// ---- VISUs/Text/InputText.TcTLO
TEXTLIST InputText
  0 = 'IN00 启动' | Chinese: 'IN00 启动' | English: 'IN00 Start' | Vietnamese: 'IN00 Kh?i ??ng ?'
  1 = 'IN01 停止' | Chinese: 'IN01 停止' | English: 'IN01 Stop' | Vietnamese: 'IN01 D?ng l?i ?'
  2 = 'IN02 复位' | Chinese: 'IN02 复位' | English: 'IN02 ResetAlarm' | Vietnamese: 'IN02 Tuy nhiên ?'
  3 = 'IN03 急停' | Chinese: 'IN03 急停' | English: 'IN03 EStop' | Vietnamese: 'IN03 V?i d?ng l?i ?'
  4 = 'IN04 安全门开关' | Chinese: 'IN04 安全门开关' | English: 'IN04 Door' | Vietnamese: 'IN04 Chuy?n ??i c?a an toàn ?'
  5 = 'IN05 工装误合盖检测光电 ' | Chinese: 'IN05 工装误合盖检测光电 ' | English: 'IN05 FrockCloseCheck' | Vietnamese: 'IN05 FrockCloseCheck'
  6 = 'IN06 解锁站流入光电' | Chinese: 'IN06 解锁站流入光电' | English: 'IN06 OpenLockCheck0' | Vietnamese: 'IN06 OpenLockCheck0'
  7 = 'IN07 预留' | Chinese: 'IN07 预留' | English: 'IN07 None3' | Vietnamese: 'IN07 Dành riêng ?'
  8 = 'IN08 主流线拨料升降气缸原位' | Chinese: 'IN08 主流线拨料升降气缸原位' | English: 'IN08 Line0PushElevator_Cyl_H' | Vietnamese: 'IN08 Line0PushElevator_Cyl_H'
  9 = 'IN09 主流线拨料升降气缸工作位' | Chinese: 'IN09 主流线拨料升降气缸工作位' | English: 'IN09 Line0PushElevator_Cyl_W' | Vietnamese: 'IN09 Line0PushElevator_Cyl_W'
  10 = 'IN0A 预留' | Chinese: 'IN0A 预留' | English: 'IN0A None6' | Vietnamese: 'IN0A Dành riêng ?'
  11 = 'IN0B 预留' | Chinese: 'IN0B 预留' | English: 'IN0B None7' | Vietnamese: 'IN0B Dành riêng ?'
  12 = 'IN0C 主流线拨料气缸安全位' | Chinese: 'IN0C 主流线拨料气缸安全位' | English: 'IN0C Line0Push_Cyl_Safe' | Vietnamese: 'IN0C Line0Push_Cyl_Safe'
  13 = 'IN0D 接驳线前阻挡光电' | Chinese: 'IN0D 接驳线前阻挡光电' | English: 'IN0D AcquireCheck3' | Vietnamese: 'IN0D AcquireCheck3'
  14 = 'IN0E 接驳线前前阻挡气缸原位' | Chinese: 'IN0E 接驳线前前阻挡气缸原位' | English: 'IN0E AcquirePrevent2_Cyl_H' | Vietnamese: 'IN0E AcquirePrevent2_Cyl_H'
  15 = 'IN0F 接驳线前前阻挡气缸工作位' | Chinese: 'IN0F 接驳线前前阻挡气缸工作位' | English: 'IN0F AcquirePrevent2_Cyl_W' | Vietnamese: 'IN0F AcquirePrevent2_Cyl_W'
  16 = 'IN10 主流线分料气缸原位' | Chinese: 'IN10 主流线分料气缸原位' | English: 'IN10 Line0Part_Cyl_H' | Vietnamese: 'IN10 Xi lanh ph?n ph?i dòng chính ?'
  17 = 'IN11 主流线分料气缸工作位' | Chinese: 'IN11 主流线分料气缸工作位' | English: 'IN11 Line0Part_Cyl_W' | Vietnamese: 'IN11 Xi lanh làm vi?c dòng chính ?'
  18 = 'IN12 主流线阻挡气缸原位' | Chinese: 'IN12 主流线阻挡气缸原位' | English: 'IN12 Line0Prevent_Cyl_H' | Vietnamese: 'IN12 Dòng chính ch?n xi lanh ?'
  19 = 'IN13 主流线阻挡气缸工作位' | Chinese: 'IN13 主流线阻挡气缸工作位' | English: 'IN13 Line0Prevent_Cyl_W' | Vietnamese: 'IN13 Dòng chính ch?n v? trí làm vi?c c?a xi lanh ?'
  20 = 'IN14 主流线拨料气缸原位' | Chinese: 'IN14 主流线拨料气缸原位' | English: 'IN14 Line0Push_Cyl_H' | Vietnamese: 'IN14 Xi lanh ?i?u ch?nh dòng chính ?'
  21 = 'IN15 主流线拨料气缸工作位' | Chinese: 'IN15 主流线拨料气缸工作位' | English: 'IN15 Line0Push_Cyl_W' | Vietnamese: 'IN15 Xi lanh dòng chính dòng v? trí làm vi?c ?'
  22 = 'IN16 接驳线前阻挡气缸原位' | Chinese: 'IN16 接驳线前阻挡气缸原位' | English: 'IN16 AcquirePrevent0_Cyl_H' | Vietnamese: 'IN16 Ch?n xi lanh tr??c d?y n?i ?'
  23 = 'IN17 接驳线前阻挡气缸工作位' | Chinese: 'IN17 接驳线前阻挡气缸工作位' | English: 'IN17 AcquirePrevent0_Cyl_W' | Vietnamese: 'IN17 Ch?n xi lanh tr??c d?y n?i ?'
  24 = 'IN18 接驳线后阻挡气缸原位' | Chinese: 'IN18 接驳线后阻挡气缸原位' | English: 'IN18 AcquirePrevent1_Cyl_H' | Vietnamese: 'IN18 Ch?n xi lanh t?i v? trí sau khi k?t n?i ?'
  25 = 'IN19 接驳线后阻挡气缸工作位' | Chinese: 'IN19 接驳线后阻挡气缸工作位' | English: 'IN19 AcquirePrevent1_Cyl_W' | Vietnamese: 'IN19 Ch?n xi lanh sau khi k?t n?i ?'
  26 = 'IN1A 接驳线顶升气缸原位' | Chinese: 'IN1A 接驳线顶升气缸原位' | English: 'IN1A AcquireLift_Cyl_H' | Vietnamese: 'IN1A Xi lanh Leo lên d?y ?i?n v? trí ?'
  27 = 'IN1B 接驳线顶升气缸工作位' | Chinese: 'IN1B 接驳线顶升气缸工作位' | English: 'IN1B AcquireLift_Cyl_W' | Vietnamese: 'IN1B Xi lanh làm vi?c trên d?y n?i ?'
  28 = 'IN1C 接驳模组拨料气缸原位' | Chinese: 'IN1C 接驳模组拨料气缸原位' | English: 'IN1C AcquirePush_Cyl_H' | Vietnamese: 'IN1C Xi lanh kh?p n?i m?-?un v? trí ?'
  29 = 'IN1D 接驳模组拨料气缸工作位' | Chinese: 'IN1D 接驳模组拨料气缸工作位' | English: 'IN1D AcquirePush_Cyl_W' | Vietnamese: 'IN1D Xi lanh làm vi?c k?t n?i m?-?un ?'
  30 = 'IN1E 接驳模组升降气缸原位' | Chinese: 'IN1E 接驳模组升降气缸原位' | English: 'IN1E AcquireElevator_Cyl_H' | Vietnamese: 'IN1E Xi lanh n?ng m?-?un k?t n?i v? trí ?'
  31 = 'IN1F 接驳模组升降气缸工作位' | Chinese: 'IN1F 接驳模组升降气缸工作位' | English: 'IN1F AcquireElevator_Cyl_W' | Vietnamese: 'IN1F K?t n?i m?-?un n?ng xi lanh v? trí làm vi?c ?'
  32 = 'IN20 转向站顶升气缸原位' | Chinese: 'IN20 转向站顶升气缸原位' | English: 'IN20 SteeringLift_Cyl_H' | Vietnamese: 'IN20 H??ng v? v? trí xi lanh n?ng lên ?'
  33 = 'IN21 转向站顶升气缸工作位' | Chinese: 'IN21 转向站顶升气缸工作位' | English: 'IN21 SteeringLift_Cyl_W' | Vietnamese: 'IN21 V? trí làm vi?c c?a xi lanh n?ng lên ?'
  34 = 'IN22 转向站接驳升降气缸原位' | Chinese: 'IN22 转向站接驳升降气缸原位' | English: 'IN22 SteeringAcquireElevator_Cyl_H' | Vietnamese: 'IN22 Chuy?n h??ng k?t n?i v?i xi lanh n?ng t?i v? trí ?'
  35 = 'IN23 转向站接驳升降气缸工作位' | Chinese: 'IN23 转向站接驳升降气缸工作位' | English: 'IN23 SteeringAcquireElevator_Cyl_W' | Vietnamese: 'IN23 Chuy?n h??ng tr?m n?i xi lanh n?ng v? trí làm vi?c ?'
  36 = 'IN24 转向站旋转气缸原位' | Chinese: 'IN24 转向站旋转气缸原位' | English: 'IN24 SteeringRotate_Cyl_H' | Vietnamese: 'IN24 Tr?m quay quay xi lanh v? trí ?'
  37 = 'IN25 转向站旋转气缸工作位' | Chinese: 'IN25 转向站旋转气缸工作位' | English: 'IN25 SteeringRotate_Cyl_W' | Vietnamese: 'IN25 Tr?m quay quay xi lanh v? trí làm vi?c ?'
  38 = 'IN26 转向站接驳限位气缸原位' | Chinese: 'IN26 转向站接驳限位气缸原位' | English: 'IN26 SteeringAcquireLimit_Cyl_H' | Vietnamese: 'IN26 Xi lanh gi?i h?n k?t n?i tr?m lái ?'
  39 = 'IN27 转向站接驳限位气缸工作位' | Chinese: 'IN27 转向站接驳限位气缸工作位' | English: 'IN27 SteeringAcquireLimit_Cyl_W' | Vietnamese: 'IN27 V? trí làm vi?c c?a xi lanh gi?i h?n k?t n?i tr?m lái ?'
  40 = 'IN28 解锁站阻挡气缸原位' | Chinese: 'IN28 解锁站阻挡气缸原位' | English: 'IN28 OpenLockPrevent_Cyl_H' | Vietnamese: 'IN28 M? khóa tr?m ?? ng?n ch?n xi lanh ?'
  41 = 'IN29 解锁站阻挡气缸工作位' | Chinese: 'IN29 解锁站阻挡气缸工作位' | English: 'IN29 OpenLockPrevent_Cyl_W' | Vietnamese: 'IN29 M? khóa tr?m ?? ch?n v? trí làm vi?c c?a xi lanh ?'
  42 = 'IN2A 解锁站顶升气缸原位' | Chinese: 'IN2A 解锁站顶升气缸原位' | English: 'IN2A OpenLockLift_Cyl_H' | Vietnamese: 'IN2A M? khóa tr?m n?ng xi lanh v? trí ?'
  43 = 'IN2B 解锁站顶升气缸工作位' | Chinese: 'IN2B 解锁站顶升气缸工作位' | English: 'IN2B OpenLockLift_Cyl_W' | Vietnamese: 'IN2B Xi lanh m? khóa tr?m làm vi?c ?'
  44 = 'IN2C 解锁站侧推气缸原位' | Chinese: 'IN2C 解锁站侧推气缸原位' | English: 'IN2C OpenLockPush_Cyl_H' | Vietnamese: 'IN2C M? khóa xi lanh ??y ga ?'
  45 = 'IN2D 解锁站侧推气缸工作位' | Chinese: 'IN2D 解锁站侧推气缸工作位' | English: 'IN2D OpenLockPush_Cyl_W' | Vietnamese: 'IN2D M? khóa v? trí làm vi?c xi lanh ??y ga ?'
  46 = 'IN2E 解锁站旋转气缸原位' | Chinese: 'IN2E 解锁站旋转气缸原位' | English: 'IN2E OpenLockRotate_Cyl_H' | Vietnamese: 'IN2E M? khóa tr?m quay xi lanh v? trí ?'
  47 = 'IN2F 解锁站旋转气缸工作位' | Chinese: 'IN2F 解锁站旋转气缸工作位' | English: 'IN2F OpenLockRotate_Cyl_W' | Vietnamese: 'IN2F Tr?m m? khóa xi lanh quay v? trí làm vi?c ?'
  48 = 'IN30 解锁站侧推气缸2原位' | Chinese: 'IN30 解锁站侧推气缸2原位' | English: 'IN30 OpenLockPush2_Cyl_H' | Vietnamese: 'IN30 M? khóa xi lanh 2 ??y ga ?'
  49 = 'IN31 解锁站侧推气缸2工作位' | Chinese: 'IN31 解锁站侧推气缸2工作位' | English: 'IN31 OpenLockPush2_Cyl_W' | Vietnamese: 'IN31 M? khóa xi lanh bên ga ??y v? trí làm vi?c 2 ?'
  50 = 'IN32 取UC站阻挡气缸原位' | Chinese: 'IN32 取UC站阻挡气缸原位' | English: 'IN32 TakeUcPrevent_Cyl_H' | Vietnamese: 'IN32 L?y tr? UC ?? ch?n xi lanh ?'
  51 = 'IN33 取UC站阻挡气缸工作位' | Chinese: 'IN33 取UC站阻挡气缸工作位' | English: 'IN33 TakeUcPrevent_Cyl_W' | Vietnamese: 'IN33 L?y v? trí làm vi?c c?a xi lanh t? tr?m UC ?'
  52 = 'IN34 取UC站顶升气缸原位' | Chinese: 'IN34 取UC站顶升气缸原位' | English: 'IN34 TakeUcLift_Cyl_H' | Vietnamese: 'IN34 L?y xi lanh n?ng lên ? tr?m UC ?'
  53 = 'IN35 取UC站顶升气缸工作位' | Chinese: 'IN35 取UC站顶升气缸工作位' | English: 'IN35 TakeUcLift_Cyl_W' | Vietnamese: 'IN35 L?y v? trí làm vi?c c?a xi lanh n?ng lên t? tr?m UC ?'
  54 = 'IN36 取UC站侧推气缸原位' | Chinese: 'IN36 取UC站侧推气缸原位' | English: 'IN36 TakeUcPush_Cyl_H' | Vietnamese: 'IN36 L?y xi lanh ??y bên ga UC ?'
  55 = 'IN37 取UC站侧推气缸工作位' | Chinese: 'IN37 取UC站侧推气缸工作位' | English: 'IN37 TakeUcPush_Cyl_W' | Vietnamese: 'IN37 L?y v? trí làm vi?c c?a xi lanh ??y bên ga UC ?'
  56 = 'IN38 取UC站旋转气缸原位' | Chinese: 'IN38 取UC站旋转气缸原位' | English: 'IN38 TakeUcRotate_Cyl_H' | Vietnamese: 'IN38 L?y xi lanh quay ? tr?m UC ?'
  57 = 'IN39 取UC站旋转气缸工作位' | Chinese: 'IN39 取UC站旋转气缸工作位' | English: 'IN39 TakeUcRotate_Cyl_W' | Vietnamese: 'IN39 L?y v? trí quay xi lanh c?a tr?m UC ?'
  58 = 'IN3A 取UC站校平气缸原位' | Chinese: 'IN3A 取UC站校平气缸原位' | English: 'IN3A TakeUcStandard_Cyl_H' | Vietnamese: 'IN3A L?y xi lanh ph?ng ? ga UC ?'
  59 = 'IN3B 取UC站校平气缸工作位' | Chinese: 'IN3B 取UC站校平气缸工作位' | English: 'IN3B TakeUcStandard_Cyl_W' | Vietnamese: 'IN3B Tr?m ki?m tra xi lanh b?ng ph?ng ?'
  60 = 'IN3C 取UC站工装夹紧气缸原位' | Chinese: 'IN3C 取UC站工装夹紧气缸原位' | English: 'IN3C TakeUcFrockClamp_Cyl_H' | Vietnamese: 'IN3C L?y xi lanh k?p vào v? trí c?a tr?m UC'
  61 = 'IN3D 取UC站工装夹紧气缸工作位' | Chinese: 'IN3D 取UC站工装夹紧气缸工作位' | English: 'IN3D TakeUcFrockClamp_Cyl_W' | Vietnamese: 'IN3D L?y v? trí làm vi?c xi lanh cài ??t ? ga UC'
  62 = 'IN3E 下工装站阻挡气缸原位' | Chinese: 'IN3E 下工装站阻挡气缸原位' | English: 'IN3E UnloadFrockPrevent_Cyl_H' | Vietnamese: 'IN3E Ng?n ch?n xi lanh ? v? trí c?ng c? ?'
  63 = 'IN3F 下工装站阻挡气缸工作位' | Chinese: 'IN3F 下工装站阻挡气缸工作位' | English: 'IN3F UnloadFrockPrevent_Cyl_W' | Vietnamese: 'IN3F Tr?m d?ng xi lanh làm vi?c ?'
  64 = 'IN40 下工装站顶升气缸原位' | Chinese: 'IN40 下工装站顶升气缸原位' | English: 'IN40 UnloadFrockLift_Cyl_H' | Vietnamese: 'IN40 Xi lanh n?ng lên xu?ng ga v? trí ?'
  65 = 'IN41 下工装站顶升气缸工作位' | Chinese: 'IN41 下工装站顶升气缸工作位' | English: 'IN41 UnloadFrockLift_Cyl_W' | Vietnamese: 'IN41 Xi lanh n?ng lên các tr?m làm vi?c ?'
  66 = 'IN42 下工装站拨料气缸原位' | Chinese: 'IN42 下工装站拨料气缸原位' | English: 'IN42 UnloadFrockPush_Cyl_H' | Vietnamese: 'IN42 Xi lanh xi lanh ? v? trí ti?p theo ?'
  67 = 'IN43 下工装站拨料气缸工作位' | Chinese: 'IN43 下工装站拨料气缸工作位' | English: 'IN43 UnloadFrockPush_Cyl_W' | Vietnamese: 'IN43 Xi lanh theo tr?m làm vi?c ?'
  68 = 'IN44 取UC模组平移Y气缸原位' | Chinese: 'IN44 取UC模组平移Y气缸原位' | English: 'IN44 TakeUc1Y_Cyl_H' | Vietnamese: 'IN44 L?y m?-?un UC và chuy?n xi lanh Y vào v? trí ?'
  69 = 'IN45 取UC模组平移Y气缸工作位' | Chinese: 'IN45 取UC模组平移Y气缸工作位' | English: 'IN45 TakeUc1Y_Cyl_W' | Vietnamese: 'IN45 Thay ??i xi lanh Y b?ng m?-?un UC ?'
  70 = 'IN46 取UC模组升降Z1气缸原位' | Chinese: 'IN46 取UC模组升降Z1气缸原位' | English: 'IN46 TakeUc1Z1_Cyl_H' | Vietnamese: 'IN46 N?ng xi lanh Z1 b?ng m?-?un UC ?'
  71 = 'IN47 取UC模组升降Z1气缸工作位' | Chinese: 'IN47 取UC模组升降Z1气缸工作位' | English: 'IN47 TakeUc1Z1_Cyl_W' | Vietnamese: 'IN47 L?y m?-?un n?ng xi lanh Z1 ?'
  72 = 'IN48 取UC模组升降Z2气缸原位' | Chinese: 'IN48 取UC模组升降Z2气缸原位' | English: 'IN48 TakeUc1Z2_Cyl_H' | Vietnamese: 'IN48 L?y m?-?un UC n?ng xi lanh Z2 ?'
  73 = 'IN49 取UC模组升降Z2气缸工作位' | Chinese: 'IN49 取UC模组升降Z2气缸工作位' | English: 'IN49 TakeUc1Z2_Cyl_W' | Vietnamese: 'IN49 L?y m?-?un UC n?ng xi lanh Z2 v? trí làm vi?c ?'
  74 = 'IN4A 取UC模组旋转气缸原位' | Chinese: 'IN4A 取UC模组旋转气缸原位' | English: 'IN4A TakeUc1Rotate_Cyl_H' | Vietnamese: 'IN4A L?y xi lanh quay c?a m?-?un UC ?'
  75 = 'IN4B 取UC模组旋转气缸工作位' | Chinese: 'IN4B 取UC模组旋转气缸工作位' | English: 'IN4B TakeUc1Rotate_Cyl_W' | Vietnamese: 'IN4B L?y v? trí làm vi?c c?a xi lanh xoay m?-?un UC ?'
  76 = 'IN4C 取UC模组夹紧气缸原位' | Chinese: 'IN4C 取UC模组夹紧气缸原位' | English: 'IN4C TakeUc1Clamp_Cyl_H' | Vietnamese: 'IN4C L?y m?-?un UC k?p xi lanh vào v? trí ?'
  77 = 'IN4D 取UC模组夹紧气缸工作位' | Chinese: 'IN4D 取UC模组夹紧气缸工作位' | English: 'IN4D TakeUc1Clamp_Cyl_W' | Vietnamese: 'IN4D L?y m?-?un UC k?p xi lanh vào v? trí làm vi?c ?'
  78 = 'IN4E 下UC皮带升降气缸原位' | Chinese: 'IN4E 下UC皮带升降气缸原位' | English: 'IN4E UnloadUcElevator_Cyl_H' | Vietnamese: 'IN4E Xi lanh n?ng d??i vành ?ai UC ?'
  79 = 'IN4F 下UC皮带升降气缸工作位' | Chinese: 'IN4F 下UC皮带升降气缸工作位' | English: 'IN4F UnloadUcElevator_Cyl_W' | Vietnamese: 'IN4F V? trí làm vi?c c?a xi lanh n?ng d??i vành ?ai UC ?'
  80 = 'IN50 下UC皮带拨料气缸原位' | Chinese: 'IN50 下UC皮带拨料气缸原位' | English: 'IN50 UnloadUcConveyorPush_Cyl_H' | Vietnamese: 'IN50 Xi lanh ?i?u ch?nh d??i vành ?ai UC ?'
  81 = 'IN51 下UC皮带拨料气缸工作位' | Chinese: 'IN51 下UC皮带拨料气缸工作位' | English: 'IN51 UnloadUcConveyorPush_Cyl_W' | Vietnamese: 'IN51 Xi lanh làm vi?c d??i vành ?ai UC ?'
  82 = 'IN52 下工装皮带升降气缸原位' | Chinese: 'IN52 下工装皮带升降气缸原位' | English: 'IN52 UnloadFrockConveyorPrevent_Cyl_H' | Vietnamese: 'IN52 D?y chuy?n n?ng xi lanh cài ??t ?'
  83 = 'IN53 下工装皮带升降气缸工作位' | Chinese: 'IN53 下工装皮带升降气缸工作位' | English: 'IN53 UnloadFrockConveyorPrevent_Cyl_W' | Vietnamese: 'IN53 D?y chuy?n n?ng xi lanh làm vi?c ?'
  84 = 'IN54 下工装皮带拨料气缸原位' | Chinese: 'IN54 下工装皮带拨料气缸原位' | English: 'IN54 UnloadFrockConveyorPush_Cyl_H' | Vietnamese: 'IN54 Xi lanh d?y chuy?n theo v? trí ?'
  85 = 'IN55 下工装皮带拨料气缸工作位' | Chinese: 'IN55 下工装皮带拨料气缸工作位' | English: 'IN55 UnloadFrockConveyorPush_Cyl_W' | Vietnamese: 'IN55 Xi lanh d?y chuy?n làm vi?c ?'
  86 = 'IN56 解锁站解压侧推气缸原位' | Chinese: 'IN56 解锁站解压侧推气缸原位' | English: 'IN56 OpenLockPressPush_Cyl_H' | Vietnamese: 'IN56 OpenLockPressPush_Cyl_H'
  87 = 'IN57 解锁站解压侧推气缸工作位' | Chinese: 'IN57 解锁站解压侧推气缸工作位' | English: 'IN57 OpenLockPressPush_Cyl_W' | Vietnamese: 'IN57 OpenLockPressPush_Cyl_W'
  88 = 'IN58 解锁站解压旋转气缸原位' | Chinese: 'IN58 解锁站解压旋转气缸原位' | English: 'IN58 OpenLockPressRotate_Cyl_H' | Vietnamese: 'IN58 OpenLockPressRotate_Cyl_H'
  89 = 'IN59 解锁站解压旋转气缸工作位' | Chinese: 'IN59 解锁站解压旋转气缸工作位' | English: 'IN59 OpenLockPressRotate_Cyl_W' | Vietnamese: 'IN59 OpenLockPressRotate_Cyl_W'
  90 = 'IN5A 预留' | Chinese: 'IN5A 预留' | English: 'IN5A None34' | Vietnamese: 'IN5A Dành riêng ?'
  91 = 'IN5B 预留' | Chinese: 'IN5B 预留' | English: 'IN5B None35' | Vietnamese: 'IN5B Dành riêng ?'
  92 = 'IN5C 下UC皮带翻转气缸缩回' | Chinese: 'IN5C 下UC皮带翻转气缸缩回' | English: 'IN5C UnloadUcBeltTipper_Cyl_H' | Vietnamese: 'IN5C Quay ng??c xi lanh l?i ?'
  93 = 'IN5D 下UC皮带翻转气缸伸出' | Chinese: 'IN5D 下UC皮带翻转气缸伸出' | English: 'IN5D UnloadUcBeltTipper_Cyl_W' | Vietnamese: 'IN5D Cái xi lanh xoay d??i vành ?ai UC thò ra ?'
  94 = 'IN5E 下UC皮带顶升气缸缩回' | Chinese: 'IN5E 下UC皮带顶升气缸缩回' | English: 'IN5E UnloadUcBeltLift_Cyl_H' | Vietnamese: 'IN5E Co l?i xi lanh n?ng lên d??i vành ?ai UC ?'
  95 = 'IN5F 下UC皮带顶升气缸伸出' | Chinese: 'IN5F 下UC皮带顶升气缸伸出' | English: 'IN5F UnloadUcBeltLift_Cyl_W' | Vietnamese: 'IN5F Cái xi lanh n?ng lên d??i vành ?ai UC thò ra ?'
  96 = 'IN60 主流线分料光电' | Chinese: 'IN60 主流线分料光电' | English: 'IN60 Line0Check1' | Vietnamese: 'IN60 Dòng chính ph?n ph?i quang ?i?n ?'
  97 = 'IN61 主流线阻挡光电' | Chinese: 'IN61 主流线阻挡光电' | English: 'IN61 Line0Check2' | Vietnamese: 'IN61 Dòng chính ng?n ch?n quang ?i?n ?'
  98 = 'IN62 主流线到位光电' | Chinese: 'IN62 主流线到位光电' | English: 'IN62 Line0Check3' | Vietnamese: 'IN62 Dòng chính vào v? trí quang ?i?n ?'
  99 = 'IN63 接驳线流入光电' | Chinese: 'IN63 接驳线流入光电' | English: 'IN63 AcquireCheck1' | Vietnamese: 'IN63 ???ng d?n d?n vào quang ?i?n ?'
  100 = 'IN64 接驳线到位光电' | Chinese: 'IN64 接驳线到位光电' | English: 'IN64 AcquireCheck2' | Vietnamese: 'IN64 K?t n?i ??n v? trí quang ?i?n ?'
  101 = 'IN65 转向站到位光电' | Chinese: 'IN65 转向站到位光电' | English: 'IN65 SteeringCheck1' | Vietnamese: 'IN65 Chuy?n sang v? trí quang ?i?n ?'
  102 = 'IN66 解锁站到位光电' | Chinese: 'IN66 解锁站到位光电' | English: 'IN66 OpenLockCheck' | Vietnamese: 'IN66 M? khóa v? trí quang ?i?n ?'
  103 = 'IN67 取UC站到位光电' | Chinese: 'IN67 取UC站到位光电' | English: 'IN67 TakeUcCheck1' | Vietnamese: 'IN67 Cho tr?m n?ng l??ng m?t tr?i vào v? trí ?'
  104 = 'IN68 下工装站到位光电' | Chinese: 'IN68 下工装站到位光电' | English: 'IN68 UnloadFrockCheck1' | Vietnamese: 'IN68 Thi?t b? ??t t?i v? trí quang ?i?n ?'
  105 = 'IN69 下UC皮带流入光电' | Chinese: 'IN69 下UC皮带流入光电' | English: 'IN69 UnloadUcCheck1' | Vietnamese: 'IN69 Vành ?ai d??i UC ?ang ch?y vào quang ?i?n ?'
  106 = 'IN6A 下UC皮带到位光电' | Chinese: 'IN6A 下UC皮带到位光电' | English: 'IN6A UnloadUcCheck2' | Vietnamese: 'IN6A Phía d??i vành ?ai n?ng l??ng m?t tr?i ?'
  107 = 'IN6B 下工装站流入光电' | Chinese: 'IN6B 下工装站流入光电' | English: 'IN6B UnloadFrockStationCheck1' | Vietnamese: 'IN6B Vành ?ai c?ng c? ch?y vào quang ?i?n ?'
  108 = 'IN6C 下工装皮带到位光电' | Chinese: 'IN6C 下工装皮带到位光电' | English: 'IN6C UnloadFrockConveyorCheck2' | Vietnamese: 'IN6C Vành ?ai c?ng c? ? v? trí quang ?i?n ?'
  109 = 'IN6D 下uc皮带翻转光电' | Chinese: 'IN6D 下uc皮带翻转光电' | English: 'IN6D UnloadUcBeltTipper' | Vietnamese: 'IN6D ??o ng??c n?ng l??ng m?t tr?i ?'
  110 = 'IN6E 取UC站流入光电' | Chinese: 'IN6E 取UC站流入光电' | English: 'IN6E TakeUcCheck0' | Vietnamese: 'IN6E TakeUcCheck0'
  111 = 'IN6F 取UC模组平移Y气缸安全位' | Chinese: 'IN6F 取UC模组平移Y气缸安全位' | English: 'IN6F TakeUc1Y_Cyl_Safe' | Vietnamese: 'IN6F Dành riêng ?'
  112 = 'IN70 解锁站升降气缸原位' | Chinese: 'IN70 解锁站升降气缸原位' | English: 'IN70 OpenLockElevator_Cyl_H' | Vietnamese: 'IN70 M? khóa tr?m n?ng xi lanh v? trí ?'
  113 = 'IN71 解锁站升降气缸工作位' | Chinese: 'IN71 解锁站升降气缸工作位' | English: 'IN71 OpenLockElevator_Cyl_W' | Vietnamese: 'IN71 M? khóa tr?m n?ng xi lanh v? trí làm vi?c ?'
  114 = 'IN72 解锁站解锁平移原位' | Chinese: 'IN72 解锁站解锁平移原位' | English: 'IN72 OpenLockPin_Cyl_H' | Vietnamese: 'IN72 Tr?m m? khóa m? khóa chuy?n v? trí ?'
  115 = 'IN73 解锁站解锁平移工作位' | Chinese: 'IN73 解锁站解锁平移工作位' | English: 'IN73 OpenLockPin_Cyl_W' | Vietnamese: 'IN73 Tr?m m? khóa m? khóa chuy?n v? trí làm vi?c ?'
  116 = 'IN74 解锁站按压气缸到原位' | Chinese: 'IN74 解锁站按压气缸到原位' | English: 'IN74 TakeUcElevator_Cyl_H' | Vietnamese: 'IN74 M? khóa tr?m nh?n xi lanh vào v? trí ?'
  117 = 'IN75 解锁站按压气缸到工作位' | Chinese: 'IN75 解锁站按压气缸到工作位' | English: 'IN75 TakeUcElevator_Cyl_W' | Vietnamese: 'IN75 M? khóa tr?m nh?n xi lanh ??n v? trí làm vi?c ?'
  118 = 'IN76 取UC站升降气缸原位' | Chinese: 'IN76 取UC站升降气缸原位' | English: 'IN76 TakeUcPush1_Cyl_H' | Vietnamese: 'IN76 L?y xi lanh n?ng t? tr?m UC ?'
  119 = 'IN77 取UC站升降气缸工作位' | Chinese: 'IN77 取UC站升降气缸工作位' | English: 'IN77 TakeUcPush1_Cyl_W' | Vietnamese: 'IN77 Tr? UC n?ng xi lanh v? trí làm vi?c ?'
  120 = 'IN78 取UC站侧推1气缸到原位' | Chinese: 'IN78 取UC站侧推1气缸到原位' | English: 'IN78 None45' | Vietnamese: 'IN78 L?y ga UC ??y 1 xi lanh vào v? trí ?'
  121 = 'IN79 取UC站侧推1气缸到工作位' | Chinese: 'IN79 取UC站侧推1气缸到工作位' | English: 'IN79 None46' | Vietnamese: 'IN79 L?y ga bên ??y 1 xi lanh t?i v? trí làm vi?c ?'
  122 = 'IN7A 预留' | Chinese: 'IN7A 预留' | English: 'IN7A None45' | Vietnamese: 'IN7A Dành riêng ?'
  123 = 'IN7B 预留' | Chinese: 'IN7B 预留' | English: 'IN7B None46' | Vietnamese: 'IN7B Dành riêng ?'
  124 = 'IN7C 预留' | Chinese: 'IN7C 预留' | English: 'IN7C None47' | Vietnamese: 'IN7C Dành riêng ?'
  125 = 'IN7D 预留' | Chinese: 'IN7D 预留' | English: 'IN7D None48' | Vietnamese: 'IN7D Dành riêng ?'
  126 = 'IN7E 预留' | Chinese: 'IN7E 预留' | English: 'IN7E None49' | Vietnamese: 'IN7E Dành riêng ?'
  127 = 'IN7F 预留' | Chinese: 'IN7F 预留' | English: 'IN7F None50' | Vietnamese: 'IN7F Dành riêng ?'
   = ''
END_TEXTLIST

// ---- VISUs/Text/LineLoadClose.TcTLO
TEXTLIST LineLoadClose
  0 = '主流线&缓存线上料' | Chinese: '主流线&缓存线上料' | English: 'LineLoad_None' | Vietnamese: 'LineLoad_None'
  1 = '主流线上料关闭' | Chinese: '主流线上料关闭' | English: 'Line0Close' | Vietnamese: 'Line1Close'
  2 = '缓存线上料关闭' | Chinese: '缓存线上料关闭' | English: 'LineAcquireClose' | Vietnamese: 'LineAcquireClose'
   = ''
END_TEXTLIST

// ---- VISUs/Text/LineLoadClase.TcTLO
TEXTLIST LineLoadClase
  0 = '不选择' | Chinese: '不选择' | English: 'None' | Vietnamese: 'None'
  1 = '优先主流线' | Chinese: '优先主流线' | English: 'Priority Line0' | Vietnamese: 'Priority Line0'
  2 = '优先接驳站' | Chinese: '优先接驳站' | English: 'Priority Acquire' | Vietnamese: 'Priority Acquire'
  3 = '优先传感器' | Chinese: '优先传感器' | English: 'Priority Sensor' | Vietnamese: 'Priority Sensor'
   = ''
END_TEXTLIST

// ---- VISUs/Text/LoadPriority.TcTLO
TEXTLIST LoadPriority
  0 = 'LoadPriority_None'
  1 = 'LoadPriority_Line0'
  2 = 'LoadPriority_Line1'
   = ''
END_TEXTLIST

// ---- VISUs/Text/MachineType.TcTLO
TEXTLIST MachineType
  0 = 'None'
  1 = '367' | Chinese: '367' | English: '367' | Vietnamese: '367'
  2 = '201' | Chinese: '201' | English: '201' | Vietnamese: '201'
  3 = '373' | Chinese: '373' | English: '373' | Vietnamese: '373'
  4 = '69' | Chinese: '69' | English: '69' | Vietnamese: '69'
  5 = '311' | Chinese: '311' | English: '311' | Vietnamese: '311'
   = ''
END_TEXTLIST

// ---- VISUs/Text/ProductType.TcTLO
TEXTLIST ProductType
  0 = '无' | Chinese: '无' | English: 'None' | Vietnamese: 'None'
  1 = '左线' | Chinese: '左线' | English: 'Left' | Vietnamese: 'Left'
  2 = '右线' | Chinese: '右线' | English: 'Right' | Vietnamese: 'Right'
   = ''
END_TEXTLIST

// ---- VISUs/Text/ManualText.TcTLO
TEXTLIST ManualText
  0 = ' \n  取料Y轴\n1:初始位 2:Line0取料位 3:Line1取料位 4:Line3取料位\n\n   取料Z轴\n1:上升位 2:下降位_Line0 3:下降位_Line1\n\n   下UC_Y轴\n1:初始位 2:Line2取料位 3:Line3取料位 4:下UC位' | Chinese: ' \n  取料Y轴\n1:初始位 2:Line0取料位 3:Line1取料位 4:Line3取料位\n\n   取料Z轴\n1:上升位 2:下降位_Line0 3:下降位_Line1\n\n   下UC_Y轴\n1:初始位 2:Line2取料位 3:Line3取料位 4:下UC位' | English: ' \nPick the y axis\nThe initial bit is the initial bit 2:line0\n\nPick the z axis\nDrop _line0 3: drop _line1\n\nThe lower uc_y axis\n1: the initial bit 2:line2 takes the material bit \n3:line3 takes the material bit 4: the lower uc bit' | Vietnamese: ' \nL?y v?t li?u trên tr?c Y\n1: ban ??u bit 2: dòng 0 c?p 3: dòng 1 c?p 4: dòng 3 c?p\n\nL?y tr?c Z\n1: n?ng lên 2: h? xu?ng bit _dòng 0 3: h? xu?ng bit _dòng 1\n\nTr?c d??i UC_Y\n1: b?t ??u bit 2: dòng 2 c?p 3: dòng 3 c?p 4: UC'
   = ''
END_TEXTLIST

// ---- VISUs/Text/OutputText.TcTLO
TEXTLIST OutputText
  0 = 'OUT00 三色灯红' | Chinese: 'OUT00 三色灯红' | English: 'OUT00 Beacon_Red' | Vietnamese: 'OUT00 ?èn ?? ba màu ?'
  1 = 'OUT01 三色灯黄' | Chinese: 'OUT01 三色灯黄' | English: 'OUT01 Beacon_Yellow' | Vietnamese: 'OUT01 ?èn màu vàng ?'
  2 = 'OUT02 三色灯绿' | Chinese: 'OUT02 三色灯绿' | English: 'OUT02 Beacon_Green' | Vietnamese: 'OUT02 Màu xanh lá c?y ?èn ba màu ?'
  3 = 'OUT03 蜂鸣器' | Chinese: 'OUT03 蜂鸣器' | English: 'OUT03 Beacon_Buzzer' | Vietnamese: 'OUT03 buzzer ?'
  4 = 'OUT04 运行指示灯' | Chinese: 'OUT04 运行指示灯' | English: 'OUT04 Runing' | Vietnamese: 'OUT04 Ch?y ánh sáng ?'
  5 = 'OUT05 停止指示灯' | Chinese: 'OUT05 停止指示灯' | English: 'OUT05 Stop' | Vietnamese: 'OUT05 D?ng ?èn ?'
  6 = 'OUT06 照明灯' | Chinese: 'OUT06 照明灯' | English: 'OUT06 LED' | Vietnamese: 'OUT06 ?nh sáng ?'
  7 = 'OUT07 预留' | Chinese: 'OUT07 预留' | English: 'OUT07 None1' | Vietnamese: 'OUT07 Dành riêng ?'
  8 = 'OUT08 解锁站解压侧推气缸到原位' | Chinese: 'OUT08 解锁站解压侧推气缸到原位' | English: 'OUT08 OpenLockPressPush_Cyl_H' | Vietnamese: 'OUT08 OpenLockPressPush_Cyl_H'
  9 = 'OUT09 解锁站解压侧推气缸到工作位' | Chinese: 'OUT09 解锁站解压侧推气缸到工作位' | English: 'OUT09 OpenLockPressPush_Cyl_W' | Vietnamese: 'OUT09 OpenLockPressPush_Cyl_W'
  10 = 'OUT0A 解锁站解压旋转气缸到原位' | Chinese: 'OUT0A 解锁站解压旋转气缸到原位' | English: 'OUT0A OpenLockPressRotate_Cyl_H' | Vietnamese: 'OUT0A OpenLockPressRotate_Cyl_H'
  11 = 'OUT0B 解锁站解压旋转气缸到工作位' | Chinese: 'OUT0B 解锁站解压旋转气缸到工作位' | English: 'OUT0B OpenLockPressRotate_Cyl_W' | Vietnamese: 'OUT0B OpenLockPressRotate_Cyl_W'
  12 = 'OUT0C 主流线拨料升降气缸到原位' | Chinese: 'OUT0C 主流线拨料升降气缸到原位' | English: 'OUT0C Line0PushElevator_Cyl_H' | Vietnamese: 'OUT0C Line0PushElevator_Cyl_H'
  13 = 'OUT0D 主流线拨料升降气缸到工作位' | Chinese: 'OUT0D 主流线拨料升降气缸到工作位' | English: 'OUT0D Line0PushElevator_Cyl_W' | Vietnamese: 'OUT0D Line0PushElevator_Cyl_W'
  14 = 'OUT0E 接驳线前前阻挡气缸缩回' | Chinese: 'OUT0E 接驳线前前阻挡气缸缩回' | English: 'OUT0E AcquirePrevent2_Cyl_H' | Vietnamese: 'OUT0E AcquirePrevent2_Cyl_H'
  15 = 'OUT0F 接驳线前前阻挡气缸伸出' | Chinese: 'OUT0F 接驳线前前阻挡气缸伸出' | English: 'OUT0F AcquirePrevent2_Cyl_W' | Vietnamese: 'OUT0F AcquirePrevent2_Cyl_W'
  16 = 'OUT10 主流线分料气缸缩回' | Chinese: 'OUT10 主流线分料气缸缩回' | English: 'OUT10 Line0Part_Cyl_H' | Vietnamese: 'OUT10 Xi lanh c?a dòng chính rút lui ?'
  17 = 'OUT11 主流线分料气缸伸出' | Chinese: 'OUT11 主流线分料气缸伸出' | English: 'OUT11 Line0Part_Cyl_W' | Vietnamese: 'OUT11 Xi lanh dòng chính ra ngoài ?'
  18 = 'OUT12 主流线阻挡气缸缩回' | Chinese: 'OUT12 主流线阻挡气缸缩回' | English: 'OUT12 Line0Prevent_Cyl_H' | Vietnamese: 'OUT12 Dòng chính ng?n ch?n s? rút l?i c?a xi lanh ?'
  19 = 'OUT13 主流线阻挡气缸伸出' | Chinese: 'OUT13 主流线阻挡气缸伸出' | English: 'OUT13 Line0Prevent_Cyl_W' | Vietnamese: 'OUT13 Dòng chính ng?n các xi lanh thoát ra ?'
  20 = 'OUT14 主流线拨料气缸缩回' | Chinese: 'OUT14 主流线拨料气缸缩回' | English: 'OUT14 Line0Push_Cyl_H' | Vietnamese: 'OUT14 Xi lanh quay dòng chính rút lui ?'
  21 = 'OUT15 主流线拨料气缸伸出' | Chinese: 'OUT15 主流线拨料气缸伸出' | English: 'OUT15 Line0Push_Cyl_W' | Vietnamese: 'OUT15 Xi lanh cu?n dòng chính thò ra ?'
  22 = 'OUT16 接驳线前阻挡气缸缩回' | Chinese: 'OUT16 接驳线前阻挡气缸缩回' | English: 'OUT16 AcquirePrevent0_Cyl_H' | Vietnamese: 'OUT16 Khóa xi lanh tr??c d?y n?i rút l?i ?'
  23 = 'OUT17 接驳线前阻挡气缸伸出' | Chinese: 'OUT17 接驳线前阻挡气缸伸出' | English: 'OUT17 AcquirePrevent0_Cyl_W' | Vietnamese: 'OUT17 Ch?n xi lanh tr??c d?y n?i ?'
  24 = 'OUT18 接驳线后阻挡气缸缩回' | Chinese: 'OUT18 接驳线后阻挡气缸缩回' | English: 'OUT18 AcquirePrevent1_Cyl_H' | Vietnamese: 'OUT18 Khóa xi lanh l?i sau khi k?t n?i ?'
  25 = 'OUT19 接驳线后阻挡气缸伸出' | Chinese: 'OUT19 接驳线后阻挡气缸伸出' | English: 'OUT19 AcquirePrevent1_Cyl_W' | Vietnamese: 'OUT19 Ch?n xi lanh ra sau d?y n?i ?'
  26 = 'OUT1A 接驳线顶升气缸缩回' | Chinese: 'OUT1A 接驳线顶升气缸缩回' | English: 'OUT1A AcquireLift_Cyl_H' | Vietnamese: 'OUT1A Xi lanh n?ng d?y n?i rút l?i ?'
  27 = 'OUT1B 接驳线顶升气缸伸出' | Chinese: 'OUT1B 接驳线顶升气缸伸出' | English: 'OUT1B AcquireLift_Cyl_W' | Vietnamese: 'OUT1B Xi lanh c?m trên d?y d?n ra ngoài ?'
  28 = 'OUT1C 接驳模组拨料气缸缩回' | Chinese: 'OUT1C 接驳模组拨料气缸缩回' | English: 'OUT1C AcquirePush_Cyl_H' | Vietnamese: 'OUT1C Xi lanh k?t n?i m?-?un quay l?i ?'
  29 = 'OUT1D 接驳模组拨料气缸伸出' | Chinese: 'OUT1D 接驳模组拨料气缸伸出' | English: 'OUT1D AcquirePush_Cyl_W' | Vietnamese: 'OUT1D Xi lanh k?t n?i m?-?un phát ra ?'
  30 = 'OUT1E 接驳模组升降气缸缩回' | Chinese: 'OUT1E 接驳模组升降气缸缩回' | English: 'OUT1E AcquireElevator_Cyl_H' | Vietnamese: 'OUT1E Xi lanh n?ng m?-?un n?i rút l?i ?'
  31 = 'OUT1F 接驳模组升降气缸伸出' | Chinese: 'OUT1F 接驳模组升降气缸伸出' | English: 'OUT1F AcquireElevator_Cyl_W' | Vietnamese: 'OUT1F Xi lanh n?ng m?-?un n?i thò ra ?'
  32 = 'OUT20 转向站顶升气缸缩回' | Chinese: 'OUT20 转向站顶升气缸缩回' | English: 'OUT20 SteeringLift_Cyl_H' | Vietnamese: 'OUT20 Quay tr? l?i xi lanh ?'
  33 = 'OUT21 转向站顶升气缸伸出' | Chinese: 'OUT21 转向站顶升气缸伸出' | English: 'OUT21 SteeringLift_Cyl_W' | Vietnamese: 'OUT21 Các xi lanh m? ra ?'
  34 = 'OUT22 转向站接驳升降气缸缩回' | Chinese: 'OUT22 转向站接驳升降气缸缩回' | English: 'OUT22 SteeringAcquireElevator_Cyl_H' | Vietnamese: 'OUT22 Quay l?i v?i xi lanh n?ng t?i tr?m lái ?'
  35 = 'OUT23 转向站接驳升降气缸伸出' | Chinese: 'OUT23 转向站接驳升降气缸伸出' | English: 'OUT23 SteeringAcquireElevator_Cyl_W' | Vietnamese: 'OUT23 Các xi lanh n?ng ???c n?i v?i các tr?m r? ?'
  36 = 'OUT24 转向站旋转气缸缩回' | Chinese: 'OUT24 转向站旋转气缸缩回' | English: 'OUT24 SteeringRotate_Cyl_H' | Vietnamese: 'OUT24 Quay tr?m quay xi lanh ?? rút lui ?'
  37 = 'OUT25 转向站旋转气缸伸出' | Chinese: 'OUT25 转向站旋转气缸伸出' | English: 'OUT25 SteeringRotate_Cyl_W' | Vietnamese: 'OUT25 Các xi lanh xoay ? v? trí quay thò ra ?'
  38 = 'OUT26 转向站接驳限位气缸缩回' | Chinese: 'OUT26 转向站接驳限位气缸缩回' | English: 'OUT26 SteeringAcquireLimit_Cyl_H' | Vietnamese: 'OUT26 Quay l?i xi lanh gi?i h?n k?t n?i tr?m r? ?'
  39 = 'OUT27 转向站接驳限位气缸伸出' | Chinese: 'OUT27 转向站接驳限位气缸伸出' | English: 'OUT27 SteeringAcquireLimit_Cyl_W' | Vietnamese: 'OUT27 Xi lanh gi?i h?n k?t n?i v?i tr?m lái xe ???c thò ra ?'
  40 = 'OUT28 解锁站阻挡气缸缩回' | Chinese: 'OUT28 解锁站阻挡气缸缩回' | English: 'OUT28 OpenLockPrevent_Cyl_H' | Vietnamese: 'OUT28 Tr?m m? khóa ng?n ch?n s? rút lui xi lanh ?'
  41 = 'OUT29 解锁站阻挡气缸伸出' | Chinese: 'OUT29 解锁站阻挡气缸伸出' | English: 'OUT29 OpenLockPrevent_Cyl_W' | Vietnamese: 'OUT29 Tr?m m? khóa ng?n ch?n các xi lanh thò ra ?'
  42 = 'OUT2A 解锁站顶升气缸缩回' | Chinese: 'OUT2A 解锁站顶升气缸缩回' | English: 'OUT2A OpenLockLift_Cyl_H' | Vietnamese: 'OUT2A M? khóa tr?m n?ng xi lanh rút lui ?'
  43 = 'OUT2B 解锁站顶升气缸伸出' | Chinese: 'OUT2B 解锁站顶升气缸伸出' | English: 'OUT2B OpenLockLift_Cyl_W' | Vietnamese: 'OUT2B Xi lanh m? khóa tr? n?ng thò ra ?'
  44 = 'OUT2C 解锁站侧推气缸缩回' | Chinese: 'OUT2C 解锁站侧推气缸缩回' | English: 'OUT2C OpenLockPush_Cyl_H' | Vietnamese: 'OUT2C M? khóa các xi lanh ??y ga ?? rút lui ?'
  45 = 'OUT2D 解锁站侧推气缸伸出' | Chinese: 'OUT2D 解锁站侧推气缸伸出' | English: 'OUT2D OpenLockPush_Cyl_W' | Vietnamese: 'OUT2D M? khóa ga ??y xi lanh thò ra ?'
  46 = 'OUT2E 解锁站旋转气缸缩回' | Chinese: 'OUT2E 解锁站旋转气缸缩回' | English: 'OUT2E OpenLockRotate_Cyl_H' | Vietnamese: 'OUT2E M? khóa tr?m quay xi lanh rút lui ?'
  47 = 'OUT2F 解锁站旋转气缸伸出' | Chinese: 'OUT2F 解锁站旋转气缸伸出' | English: 'OUT2F OpenLockRotate_Cyl_W' | Vietnamese: 'OUT2F Xi lanh xoay ? v? trí m? khóa thò ra ?'
  48 = 'OUT30 解锁站侧推气缸2缩回' | Chinese: 'OUT30 解锁站侧推气缸2缩回' | English: 'OUT30 OpenLockPush2_Cyl_H' | Vietnamese: 'OUT30 M? khóa ga bên ??y xi lanh 2 rút lui ?'
  49 = 'OUT31 解锁站侧推气缸2伸出' | Chinese: 'OUT31 解锁站侧推气缸2伸出' | English: 'OUT31 OpenLockPush2_Cyl_W' | Vietnamese: 'OUT31 M? khóa ga ??y xi lanh 2 thò ra ?'
  50 = 'OUT32 取UC站阻挡气缸缩回' | Chinese: 'OUT32 取UC站阻挡气缸缩回' | English: 'OUT32 TakeUcPrevent_Cyl_H' | Vietnamese: 'OUT32 L?y các tr?m ng?n ch?n và rút l?i xi lanh ?'
  51 = 'OUT33 取UC站阻挡气缸伸出' | Chinese: 'OUT33 取UC站阻挡气缸伸出' | English: 'OUT33 TakeUcPrevent_Cyl_W' | Vietnamese: 'OUT33 L?y ga ng?n ch?n lít ra ?'
  52 = 'OUT34 取UC站顶升气缸缩回' | Chinese: 'OUT34 取UC站顶升气缸缩回' | English: 'OUT34 TakeUcLift_Cyl_H' | Vietnamese: 'OUT34 L?y xi lanh n?ng lên c?a tr?m UC và rút lui ?'
  53 = 'OUT35 取UC站顶升气缸伸出' | Chinese: 'OUT35 取UC站顶升气缸伸出' | English: 'OUT35 TakeUcLift_Cyl_W' | Vietnamese: 'OUT35 L?y xi lanh n?ng lên t? tr?m UC ?'
  54 = 'OUT36 取UC站侧推气缸缩回' | Chinese: 'OUT36 取UC站侧推气缸缩回' | English: 'OUT36 TakeUcPush_Cyl_H' | Vietnamese: 'OUT36 L?y xi lanh ??y bên tàu và rút lui ?'
  55 = 'OUT37 取UC站侧推气缸伸出' | Chinese: 'OUT37 取UC站侧推气缸伸出' | English: 'OUT37 TakeUcPush_Cyl_W' | Vietnamese: 'OUT37 L?y ga bên ??y ra kh?i xi lanh ?'
  56 = 'OUT38 取UC站旋转气缸缩回' | Chinese: 'OUT38 取UC站旋转气缸缩回' | English: 'OUT38 TakeUcRotate_Cyl_H' | Vietnamese: 'OUT38 L?y xi lanh quay ? tr?m UC và rút lui ?'
  57 = 'OUT39 取UC站旋转气缸伸出' | Chinese: 'OUT39 取UC站旋转气缸伸出' | English: 'OUT39 TakeUcRotate_Cyl_W' | Vietnamese: 'OUT39 L?y các xi lanh quay t? tr?m UC ?'
  58 = 'OUT3A 取UC站校平气缸原位' | Chinese: 'OUT3A 取UC站校平气缸原位' | English: 'OUT3A TakeUcStandard_Cyl_H' | Vietnamese: 'OUT3A L?y xi lanh ph?ng ? ga UC ?'
  59 = 'OUT3B 取UC站校平气缸工作位' | Chinese: 'OUT3B 取UC站校平气缸工作位' | English: 'OUT3B TakeUcStandard_Cyl_W' | Vietnamese: 'OUT3B Tr?m ki?m tra xi lanh b?ng ph?ng ?'
  60 = 'OUT3C 取UC站工装夹紧气缸原位' | Chinese: 'OUT3C 取UC站工装夹紧气缸原位' | English: 'OUT3C TakeUcFrockClamp_Cyl_H' | Vietnamese: 'OUT3C L?y xi lanh k?p vào v? trí c?a tr?m UC'
  61 = 'OUT3D 取UC站工装夹紧气缸工作位' | Chinese: 'OUT3D 取UC站工装夹紧气缸工作位' | English: 'OUT3D TakeUcFrockClamp_Cyl_W' | Vietnamese: 'OUT3D L?y v? trí làm vi?c xi lanh cài ??t ? ga UC'
  62 = 'OUT3E 下工装站阻挡气缸缩回' | Chinese: 'OUT3E 下工装站阻挡气缸缩回' | English: 'OUT3E UnloadFrockPrevent_Cyl_H' | Vietnamese: 'OUT3E Ng?n ch?n các xi lanh rút lui ?'
  63 = 'OUT3F 下工装站阻挡气缸伸出' | Chinese: 'OUT3F 下工装站阻挡气缸伸出' | English: 'OUT3F UnloadFrockPrevent_Cyl_W' | Vietnamese: 'OUT3F Ng?n ch?n các xi lanh ra ngoài ?'
  64 = 'OUT40 下工装站顶升气缸缩回' | Chinese: 'OUT40 下工装站顶升气缸缩回' | English: 'OUT40 UnloadFrockLift_Cyl_H' | Vietnamese: 'OUT40 Xi lanh n?ng xu?ng ga xu?ng rút lui ?'
  65 = 'OUT41 下工装站顶升气缸伸出' | Chinese: 'OUT41 下工装站顶升气缸伸出' | English: 'OUT41 UnloadFrockLift_Cyl_W' | Vietnamese: 'OUT41 Xi lanh n?ng lên t? tr?m t?i xu?ng ?'
  66 = 'OUT42 下工装站拨料气缸缩回' | Chinese: 'OUT42 下工装站拨料气缸缩回' | English: 'OUT42 UnloadFrockPush_Cyl_H' | Vietnamese: 'OUT42 Xi lanh xi lanh quay tr? l?i tr?m t?i xu?ng ?'
  67 = 'OUT43 下工装站拨料气缸伸出' | Chinese: 'OUT43 下工装站拨料气缸伸出' | English: 'OUT43 UnloadFrockPush_Cyl_W' | Vietnamese: 'OUT43 Xi lanh ngu?n l?c ti?p theo ?'
  68 = 'OUT44 取UC模组平移Y气缸缩回' | Chinese: 'OUT44 取UC模组平移Y气缸缩回' | English: 'OUT44 TakeUc1Y_Cyl_H' | Vietnamese: 'OUT44 L?y m?-?un UC chuy?n xi lanh Y và rút lui ?'
  69 = 'OUT45 取UC模组平移Y气缸伸出' | Chinese: 'OUT45 取UC模组平移Y气缸伸出' | English: 'OUT45 TakeUc1Y_Cyl_W' | Vietnamese: 'OUT45 L?y m?-?un UC và di chuy?n xi lanh Y ra ngoài ?'
  70 = 'OUT46 取UC模组升降Z1气缸缩回' | Chinese: 'OUT46 取UC模组升降Z1气缸缩回' | English: 'OUT46 TakeUc1Z1_Cyl_H' | Vietnamese: 'OUT46 L?y m?-?un UC n?ng xi lanh Z1 ?? rút lui ?'
  71 = 'OUT47 取UC模组升降Z1气缸伸出' | Chinese: 'OUT47 取UC模组升降Z1气缸伸出' | English: 'OUT47 TakeUc1Z1_Cyl_W' | Vietnamese: 'OUT47 N?ng xi lanh ra kh?i m?-?un UC ?'
  72 = 'OUT48 取UC模组升降Z2气缸缩回' | Chinese: 'OUT48 取UC模组升降Z2气缸缩回' | English: 'OUT48 TakeUc1Z2_Cyl_H' | Vietnamese: 'OUT48 L?y m?-?un UC n?ng xi lanh Z2 ?? rút lui ?'
  73 = 'OUT49 取UC模组升降Z2气缸伸出' | Chinese: 'OUT49 取UC模组升降Z2气缸伸出' | English: 'OUT49 TakeUc1Z2_Cyl_W' | Vietnamese: 'OUT49 ??a ?ng n?ng Z2 ra kh?i m?-?un UC ?'
  74 = 'OUT4A 取UC模组旋转气缸缩回' | Chinese: 'OUT4A 取UC模组旋转气缸缩回' | English: 'OUT4A TakeUc1Rotate_Cyl_H' | Vietnamese: 'OUT4A Thu h?i xi lanh quay b?ng m?-?un UC ?'
  75 = 'OUT4B 取UC模组旋转气缸伸出' | Chinese: 'OUT4B 取UC模组旋转气缸伸出' | English: 'OUT4B TakeUc1Rotate_Cyl_W' | Vietnamese: 'OUT4B L?y m?-?un UC xoay xi lanh ra ngoài ?'
  76 = 'OUT4C 取UC模组夹紧气缸缩回' | Chinese: 'OUT4C 取UC模组夹紧气缸缩回' | English: 'OUT4C TakeUc1Clamp_Cyl_H' | Vietnamese: 'OUT4C L?y m?-?un UC k?p xi lanh ?? rút lui ?'
  77 = 'OUT4D 取UC模组夹紧气缸伸出' | Chinese: 'OUT4D 取UC模组夹紧气缸伸出' | English: 'OUT4D TakeUc1Clamp_Cyl_W' | Vietnamese: 'OUT4D L?y m?-?un và k?p ?ng ra ?'
  78 = 'OUT4E 下UC皮带升降气缸缩回' | Chinese: 'OUT4E 下UC皮带升降气缸缩回' | English: 'OUT4E UnloadUcElevator_Cyl_H' | Vietnamese: 'OUT4E Thu h?i xi lanh n?ng d??i vành ?ai UC ?'
  79 = 'OUT4F 下UC皮带升降气缸伸出' | Chinese: 'OUT4F 下UC皮带升降气缸伸出' | English: 'OUT4F UnloadUcElevator_Cyl_W' | Vietnamese: 'OUT4F Xi lanh n?ng d??i vành ?ai UC thò ra ?'
  80 = 'OUT50 下UC皮带拨料气缸缩回' | Chinese: 'OUT50 下UC皮带拨料气缸缩回' | English: 'OUT50 UnloadUcConveyorPush_Cyl_H' | Vietnamese: 'OUT50 Quay l?i xi lanh quay d??i vành ?ai UC ?'
  81 = 'OUT51 下UC皮带拨料气缸伸出' | Chinese: 'OUT51 下UC皮带拨料气缸伸出' | English: 'OUT51 UnloadUcConveyorPush_Cyl_W' | Vietnamese: 'OUT51 Cái xi lanh d??i vành ?ai UC thò ra ?'
  82 = 'OUT52 下工装皮带升降气缸缩回' | Chinese: 'OUT52 下工装皮带升降气缸缩回' | English: 'OUT52 UnloadFrockConveyorPrevent_Cyl_H' | Vietnamese: 'OUT52 Th?t l?ng n?ng xi lanh kéo xu?ng ?'
  83 = 'OUT53 下工装皮带升降气缸伸出' | Chinese: 'OUT53 下工装皮带升降气缸伸出' | English: 'OUT53 UnloadFrockConveyorPrevent_Cyl_W' | Vietnamese: 'OUT53 Xi lanh n?ng vành ?ai c?ng vi?c thò ra ?'
  84 = 'OUT54 下工装皮带拨料气缸缩回' | Chinese: 'OUT54 下工装皮带拨料气缸缩回' | English: 'OUT54 UnloadFrockConveyorPush_Cyl_H' | Vietnamese: 'OUT54 ?óng gói vành ?ai xi lanh quay l?i ?'
  85 = 'OUT55 下工装皮带拨料气缸伸出' | Chinese: 'OUT55 下工装皮带拨料气缸伸出' | English: 'OUT55 UnloadFrockConveyorPush_Cyl_W' | Vietnamese: 'OUT55 Xi lanh vành ?ai c?ng c? thò ra ?'
  86 = 'OUT56 接驳线前步进' | Chinese: 'OUT56 接驳线前步进' | English: 'OUT56 AcquireFrontAxis' | Vietnamese: 'OUT56 AcquireFrontAxis'
  87 = 'OUT57 接驳线步进' | Chinese: 'OUT57 接驳线步进' | English: 'OUT57 AcquireAxis' | Vietnamese: 'OUT57 B??c trên d?y n?i ?'
  88 = 'OUT58 拆解线步进' | Chinese: 'OUT58 拆解线步进' | English: 'OUT58 DismantlingAxis' | Vietnamese: 'OUT58 B??c c?t d?y ?'
  89 = 'OUT59 下UC皮带步进' | Chinese: 'OUT59 下UC皮带步进' | English: 'OUT59 UnloadUcAxis' | Vietnamese: 'OUT59 B??c xu?ng d??i vành ?ai UC ?'
  90 = 'OUT5A 下工装皮带步进' | Chinese: 'OUT5A 下工装皮带步进' | English: 'OUT5A UnloadFrock' | Vietnamese: 'OUT5A D?y n?t di chuy?n ?'
  91 = 'OUT5B 预留' | Chinese: 'OUT5B 预留' | English: 'OUT5B None21' | Vietnamese: 'OUT5B Dành riêng ?'
  92 = 'OUT5C 下UC皮带翻转气缸缩回' | Chinese: 'OUT5C 下UC皮带翻转气缸缩回' | English: 'OUT5C UnloadUcBeltTipper_Cyl_H' | Vietnamese: 'OUT5C Quay ng??c xi lanh l?i ?'
  93 = 'OUT5D 下UC皮带翻转气缸伸出' | Chinese: 'OUT5D 下UC皮带翻转气缸伸出' | English: 'OUT5D UnloadUcBeltTipper_Cyl_W' | Vietnamese: 'OUT5D Cái xi lanh xoay d??i vành ?ai UC thò ra ?'
  94 = 'OUT5E 下UC皮带顶升气缸缩回' | Chinese: 'OUT5E 下UC皮带顶升气缸缩回' | English: 'OUT5E UnloadUcBeltLift_Cyl_H' | Vietnamese: 'OUT5E Co l?i xi lanh n?ng lên d??i vành ?ai UC ?'
  95 = 'OUT5F 下UC皮带顶升气缸伸出' | Chinese: 'OUT5F 下UC皮带顶升气缸伸出' | English: 'OUT5F UnloadUcBeltLift_Cyl_W' | Vietnamese: 'OUT5F Cái xi lanh n?ng lên d??i vành ?ai UC thò ra ?'
  96 = 'OUT60 解锁站升降气缸原位' | Chinese: 'OUT60 解锁站升降气缸原位' | English: 'OUT60 OpenLockElevator_Cyl_H' | Vietnamese: 'OUT60 M? khóa tr?m n?ng xi lanh v? trí ?'
  97 = 'OUT61 解锁站升降气缸工作位' | Chinese: 'OUT61 解锁站升降气缸工作位' | English: 'OUT61 OpenLockElevator_Cyl_W' | Vietnamese: 'OUT61 M? khóa tr?m n?ng xi lanh v? trí làm vi?c ?'
  98 = 'OUT62 解锁站解锁平移原位' | Chinese: 'OUT62 解锁站解锁平移原位' | English: 'OUT62 OpenLockTranslation_Cyl_H' | Vietnamese: 'OUT62 Tr?m m? khóa m? khóa chuy?n v? trí ?'
  99 = 'OUT63 解锁站解锁平移工作位' | Chinese: 'OUT63 解锁站解锁平移工作位' | English: 'OUT63 OpenLockTranslation_Cyl_W' | Vietnamese: 'OUT63 Tr?m m? khóa m? khóa chuy?n v? trí làm vi?c ?'
  100 = 'OUT64 解锁站按压气缸到原位' | Chinese: 'OUT64 解锁站按压气缸到原位' | English: 'OUT64 OpenLockPin_Cyl_H' | Vietnamese: 'OUT64 M? khóa tr?m nh?n xi lanh vào v? trí ?'
  101 = 'OUT65 解锁站按压气缸到工作位' | Chinese: 'OUT65 解锁站按压气缸到工作位' | English: 'OUT65 OpenLockPin_Cyl_W' | Vietnamese: 'OUT65 M? khóa tr?m nh?n xi lanh ??n v? trí làm vi?c ?'
  102 = 'OUT66 取UC站升降气缸原位' | Chinese: 'OUT66 取UC站升降气缸原位' | English: 'OUT66 TakeUcElevator_Cyl_H' | Vietnamese: 'OUT66 L?y xi lanh n?ng t? tr?m UC ?'
  103 = 'OUT67 取UC站升降气缸工作位' | Chinese: 'OUT67 取UC站升降气缸工作位' | English: 'OUT67 TakeUcElevator_Cyl_W' | Vietnamese: 'OUT67 Tr? UC n?ng xi lanh v? trí làm vi?c ?'
  104 = 'OUT68 取UC站侧推1气缸到原位' | Chinese: 'OUT68 取UC站侧推1气缸到原位' | English: 'OUT68 TakeUcPush1_Cyl_H' | Vietnamese: 'OUT68 L?y ga UC ??y 1 xi lanh vào v? trí ?'
  105 = 'OUT69 取UC站侧推1气缸到工作位' | Chinese: 'OUT69 取UC站侧推1气缸到工作位' | English: 'OUT69 TakeUcPush1_Cyl_W' | Vietnamese: 'OUT69 L?y ga bên ??y 1 xi lanh t?i v? trí làm vi?c ?'
  106 = 'OUT6A 预留' | Chinese: 'OUT6A 预留' | English: 'OUT6A None35' | Vietnamese: 'OUT6A Dành riêng ?'
  107 = 'OUT6B 预留' | Chinese: 'OUT6B 预留' | English: 'OUT6B None36' | Vietnamese: 'OUT6B Dành riêng ?'
  108 = 'OUT6C 预留' | Chinese: 'OUT6C 预留' | English: 'OUT6C None37' | Vietnamese: 'OUT6C Dành riêng ?'
  109 = 'OUT6D 预留' | Chinese: 'OUT6D 预留' | English: 'OUT6D None38' | Vietnamese: 'OUT6D Dành riêng ?'
  110 = 'OUT6E 预留' | Chinese: 'OUT6E 预留' | English: 'OUT6E None39' | Vietnamese: 'OUT6E Dành riêng ?'
  111 = 'OUT6F 预留' | Chinese: 'OUT6F 预留' | English: 'OUT6F None40' | Vietnamese: 'OUT6F Dành riêng ?'
   = ''
END_TEXTLIST

// ---- VISUs/PageSetting_OpenLock.TcVIS
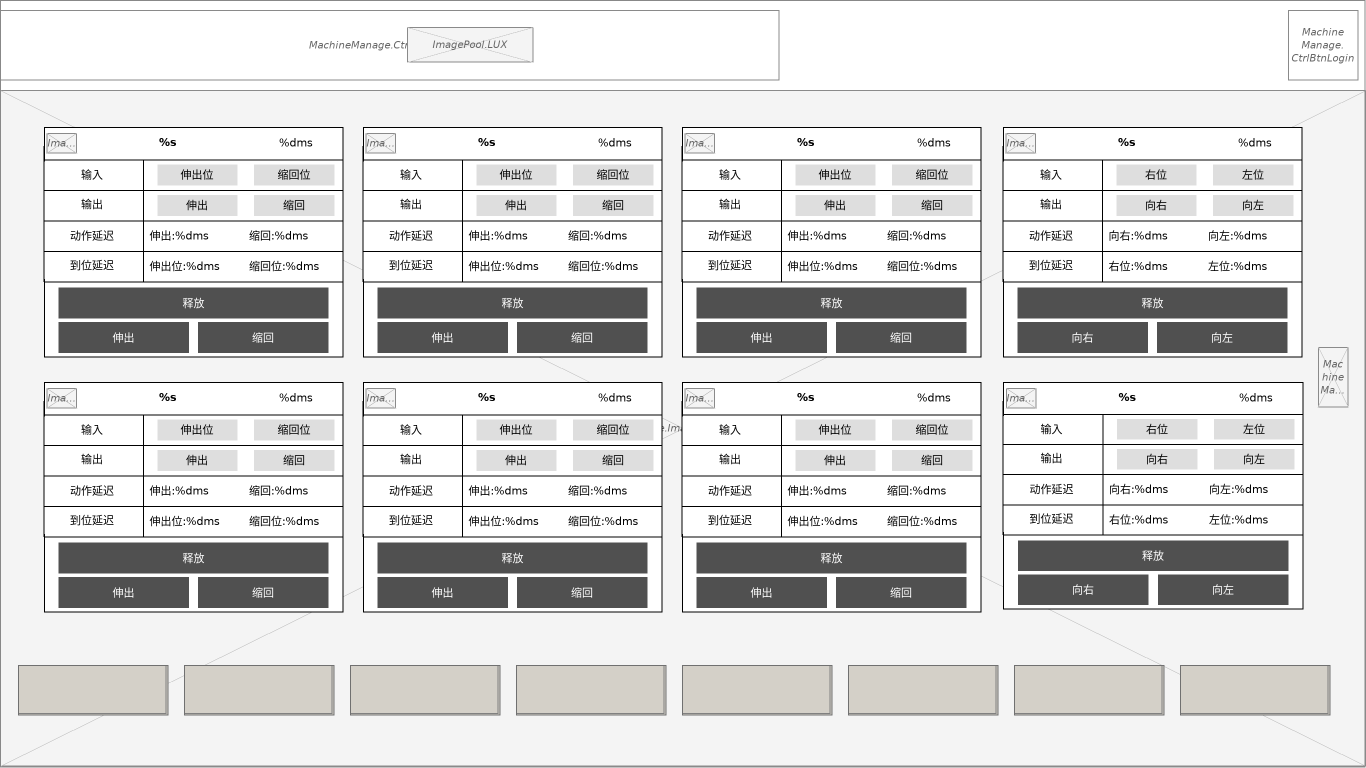
VISUALIZATION PageSetting_OpenLock  // 1366x768
    Frame (0,0 1366x768)
        shows CtrlPageSetting()
    Frame (1003,127 300x230), invisible if: GVL_Data.stRecipe.eProductType<>E_ProductType.Right or GVL_Data.stRecipe.eMachineType<> E_MachineType._311
        shows Cyliner4_1(System := G_stSystem, Cylinder := G_arrCylinder[E_Cylinder.OpenLockRotate], CylinderData := G_arrCylinderData[E_Cylinder.OpenLockRotate])
    Frame (45,127 300x230)
        shows Cyliner1(System := G_stSystem, Cylinder := G_arrCylinder[E_Cylinder.OpenLockPrevent], CylinderData := G_arrCylinderData[E_Cylinder.OpenLockPrevent])
    Frame (364,127 300x230)
        shows Cyliner1(System := G_stSystem, Cylinder := G_arrCylinder[E_Cylinder.OpenLockLift], CylinderData := G_arrCylinderData[E_Cylinder.OpenLockLift])
    Frame (683,127 300x230)
        shows Cyliner1(System := G_stSystem, Cylinder := G_arrCylinder[E_Cylinder.OpenLockPush], CylinderData := G_arrCylinderData[E_Cylinder.OpenLockPush])
    Frame (1003,127 300x230), invisible if: GVL_Data.stRecipe.eProductType<>E_ProductType.Left and GVL_Data.stRecipe.eMachineType= E_MachineType._311
        shows Cyliner4(System := G_stSystem, Cylinder := G_arrCylinder[E_Cylinder.OpenLockRotate], CylinderData := G_arrCylinderData[E_Cylinder.OpenLockRotate])
    Frame (45,382 300x230)
        shows Cyliner1(System := G_stSystem, Cylinder := G_arrCylinder[E_Cylinder.OpenLockPush2], CylinderData := G_arrCylinderData[E_Cylinder.OpenLockPush2])
    Frame (1003,382 301x227), invisible if: GVL_Data.stRecipe.eProductType<>E_ProductType.Right or GVL_Data.stRecipe.eMachineType<> E_MachineType._311
        shows Cyliner4_1(System := G_stSystem, Cylinder := G_arrCylinder[E_Cylinder.OpenLockTranslation], CylinderData := G_arrCylinderData[E_Cylinder.OpenLockTranslation])
    Frame (1003,382 301x227)
        shows Cyliner4(System := G_stSystem, Cylinder := G_arrCylinder[E_Cylinder.OpenLockTranslation], CylinderData := G_arrCylinderData[E_Cylinder.OpenLockTranslation])
    Frame (364,382 300x230)
        shows Cyliner1(System := G_stSystem, Cylinder := G_arrCylinder[E_Cylinder.OpenLockElevator], CylinderData := G_arrCylinderData[E_Cylinder.OpenLockElevator])
    Frame (683,382 300x230)
        shows Cyliner1(System := G_stSystem, Cylinder := G_arrCylinder[E_Cylinder.OpenLockPin], CylinderData := G_arrCylinderData[E_Cylinder.OpenLockPin])
    Image (1318,347 30x60), image: MachineManage.ImagePool.next
        OnMouseClick: change screen: PageSetting_OpenLock_2
END_VISUALIZATION

// ---- VISUs/PageSetting_UnloadFrock.TcVIS
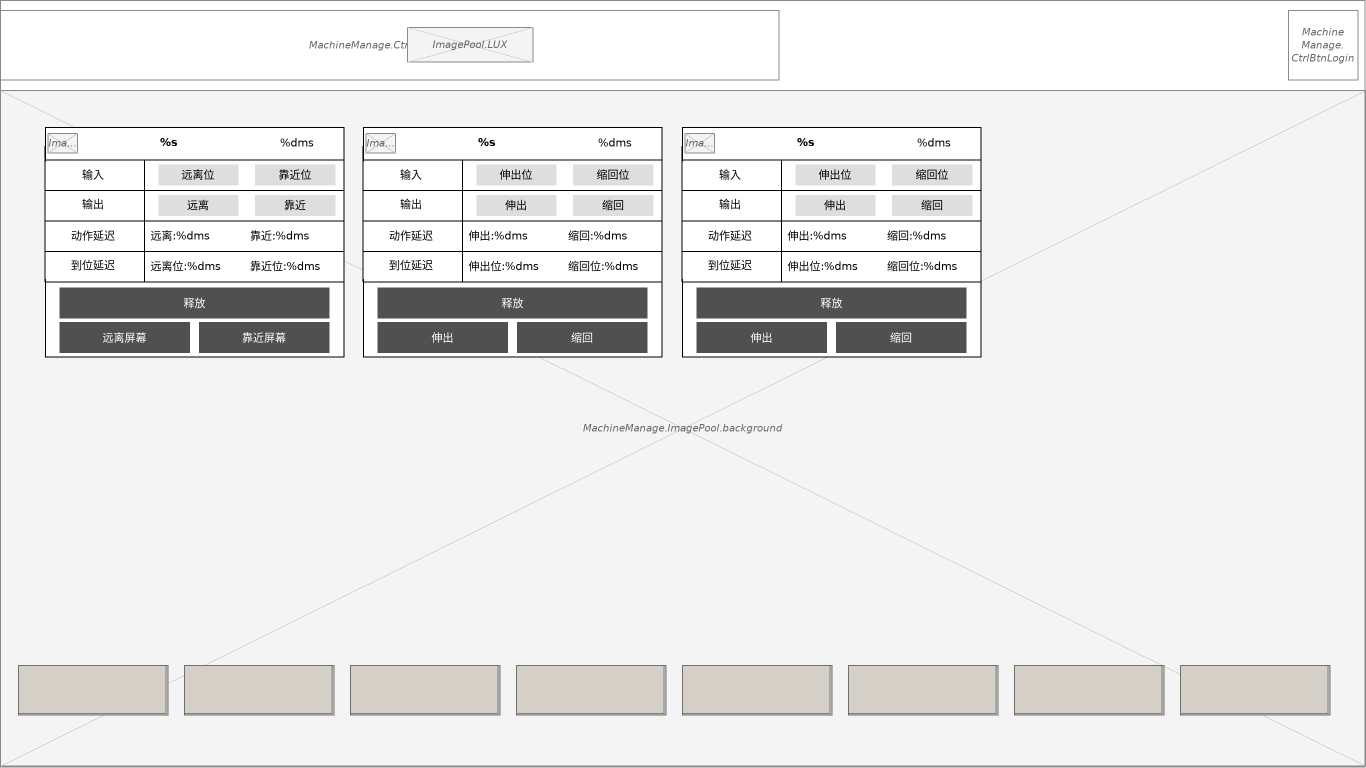
VISUALIZATION PageSetting_UnloadFrock  // 1366x768
    Frame (0,0 1366x768)
        shows CtrlPageSetting()
    Frame (683,127 300x230)
        shows Cyliner1(System := G_stSystem, Cylinder := G_arrCylinder[E_Cylinder.UnloadFrockLift], CylinderData := G_arrCylinderData[E_Cylinder.UnloadFrockLift])
    Frame (364,127 300x230)
        shows Cyliner1(System := G_stSystem, Cylinder := G_arrCylinder[E_Cylinder.UnloadFrockPrevent], CylinderData := G_arrCylinderData[E_Cylinder.UnloadFrockPrevent])
    Frame (45,127 300x230)
        shows Cyliner2(System := G_stSystem, Cylinder := G_arrCylinder[E_Cylinder.UnloadFrockPush], CylinderData := G_arrCylinderData[E_Cylinder.UnloadFrockPush])
END_VISUALIZATION

// ---- VISUs/PageSetting_TakeUc_M.TcVIS
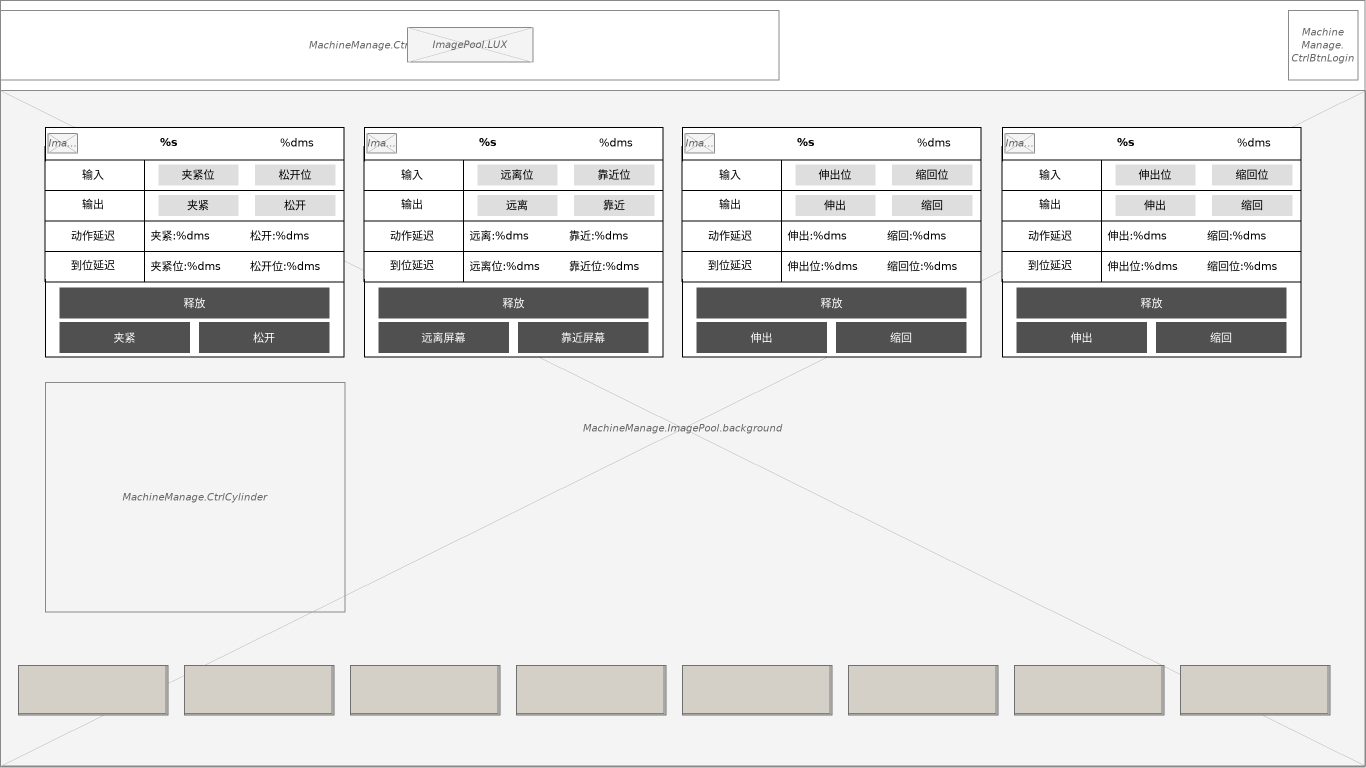
VISUALIZATION PageSetting_TakeUc_M  // 1366x768
    Frame (0,0 1366x768)
        shows CtrlPageSetting()
    Frame (364,127 300x230)
        shows Cyliner2(System := G_stSystem, Cylinder := G_arrCylinder[E_Cylinder.TakeUc1Y], CylinderData := G_arrCylinderData[E_Cylinder.TakeUc1Y])
    Frame (683,127 300x230)
        shows Cyliner1(System := G_stSystem, Cylinder := G_arrCylinder[E_Cylinder.TakeUc1Z1], CylinderData := G_arrCylinderData[E_Cylinder.TakeUc1Z1])
    Frame (1003,127 300x230)
        shows Cyliner1(System := G_stSystem, Cylinder := G_arrCylinder[E_Cylinder.TakeUc1Z2], CylinderData := G_arrCylinderData[E_Cylinder.TakeUc1Z2])
    Frame (45,382 300x230)
        shows MachineManage.CtrlCylinder(System := G_stSystem, Cylinder := G_arrCylinder[E_Cylinder.TakeUc1Rotate], CylinderData := G_arrCylinderData[E_Cylinder.TakeUc1Rotate])
    Frame (45,127 300x230)
        shows Cyliner5(System := G_stSystem, Cylinder := G_arrCylinder[E_Cylinder.TakeUc1Clamp], CylinderData := G_arrCylinderData[E_Cylinder.TakeUc1Clamp])
END_VISUALIZATION

// ---- VISUs/Text/StationName.TcTLO
TEXTLIST StationName
  0 = '接驳上料' | Chinese: '接驳上料' | English: 'AcquireLoad'
  1 = '转向站' | Chinese: '转向站' | English: 'Steering'
  2 = '解锁站' | Chinese: '解锁站' | English: 'OpenLock'
  3 = '取UC站' | Chinese: '取UC站' | English: 'TakeUc'
  4 = '取Uc模组' | Chinese: '取Uc模组' | English: 'TakeUc_M'
  5 = '下工装站' | Chinese: '下工装站' | English: 'UnloadFrock'
  6 = '下料皮带线' | Chinese: '下料皮带线' | English: 'Unload_L'
  7 = '其他' | Chinese: '其他' | English: 'Other'
   = ''
END_TEXTLIST

// ---- VISUs/PageSetting.TcVIS
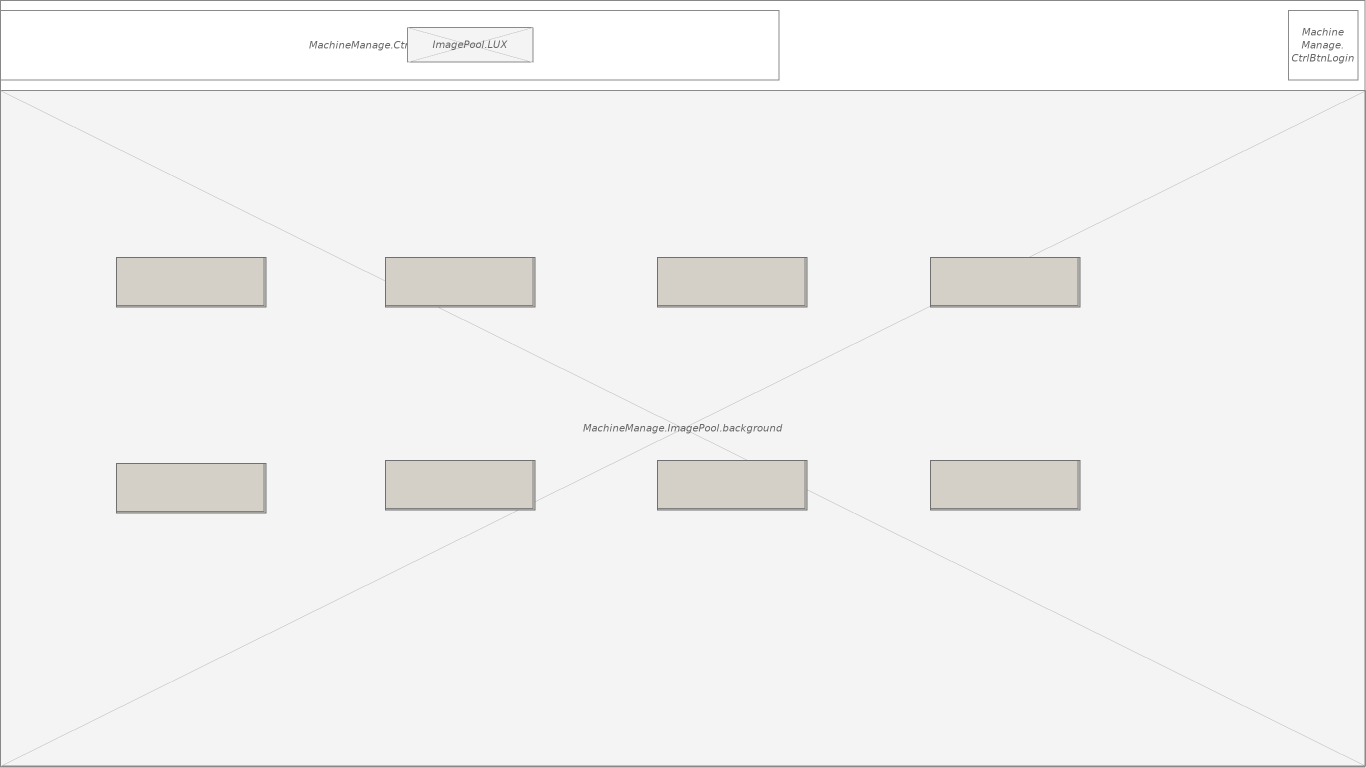
VISUALIZATION PageSetting  // 1366x768
    Frame (0,0 1366x768)
        shows FrameMain()
    Button (385,257 150x50), text list: 'StationName', text index: 1
        OnMouseClick: change screen: PageSetting_Steering
    Button (657,257 150x50), text list: 'StationName', text index: 2
        OnMouseClick: change screen: PageSetting_OpenLock
    Button (930,257 150x50), text list: 'StationName', text index: 3
        OnMouseClick: change screen: PageSetting_TakeUc
    Button (116,463 150x50), text list: 'StationName', text index: 4
        OnMouseClick: change screen: PageSetting_TakeUc_M
    Button (385,460 150x50), text list: 'StationName', text index: 5
        OnMouseClick: change screen: PageSetting_UnloadFrock
    Button (657,460 150x50), text list: 'StationName', text index: 6
        OnMouseClick: change screen: PageSetting_Unload_L
    Button (930,460 150x50), text list: 'StationName', text index: 7
        OnMouseClick: change screen: PageSetting_Other
    Button (116,257 150x50), text list: 'StationName', text index: 0
        OnMouseClick: change screen: PageSetting_AcquireLoad
END_VISUALIZATION
